{attribute 'no_explicit_call' := 'NormallyClosedPushButton is a CLASS and must be accessed using methods or properties'}
FUNCTION_BLOCK NormallyClosedPushButton implements I_PushButton
VAR
	input				AT %I*: BOOL;
END_VAR

PROPERTY IsPressed : bool
GET
IsPressed				:= not input;
END_GET
END_PROPERTY

PROPERTY IsReleased : bool
GET
IsReleased				:= input;
END_GET
END_PROPERTY

END_FUNCTION_BLOCK

(* stored: Version 1.1.0.1, ProductVersion 3.1.4024.11
   POU NormallyClosedPushButton: Id {f56c4bf2-d904-471a-ac61-ffa50c7ba15b}, SpecialFunc None
   Property IsPressed: Id {b18a6356-0fa4-455d-bf94-216ee43a5dfa}
   Get Get: Id {9805feec-4685-4d6d-ac6f-82b78d2e8bf5}
   Property IsReleased: Id {87dc275f-e4c2-48cb-aff2-a0777f240929}
   Get Get: Id {f11c0aeb-59f4-41d2-b881-2d0dcd8b724b} *)
